FUNCTION_BLOCK HeaterCatridge_control
VAR_INPUT
END_VAR
VAR_OUTPUT
END_VAR
VAR
END_VAR

END_FUNCTION_BLOCK

(* stored: Version 1.1.0.1, ProductVersion 3.1.4024.9
   POU HeaterCatridge_control: Id {dd38d42a-bd3b-456e-a2fc-9f69da39d4fa}, SpecialFunc None *)
